// TIA Portal V16 export
// export: Created 2022-07-21T09:35:15.7704888Z, ExportSetting WithDefaults, DisplayName Totally Integrated Automation Portal, DisplayVersion V16 Update 4, DisplayName TIA Portal Version Control Interface, DisplayVersion V16 Update 2, DisplayName TIA Portal Openness, DisplayVersion V16 Update 4, DisplayName SINAMICS Startdrive Advanced, DisplayVersion V16 Update 5, DisplayName SINAMICS Startdrive G130, G150, S120, S150, SINAMICS MV, S210, DisplayVersion V16 Update 5, DisplayName SINAMICS Startdrive G110M, G120, G120C, G120D, G120P, G115D, DisplayVersion V16 Update 5, DisplayName STEP 7 Professional, DisplayVersion V16 Update 4, DisplayName STEP 7 Safety, DisplayVersion V16, DisplayName WinCC Advanced, DisplayVersion V16 Update 4
DATA_BLOCK "LAxisBasics_InterfaceHMI_3"   // DB843
{ S7_Optimized_Access := 'TRUE' }
AUTHOR : ArSc
FAMILY : LAxisBasics
VERSION : 1.1
// stored: AutoNumber false, DBAccessibleFromOPCUA true, InstanceOfName LAxisBasics_typeInterfaceHMI, InstanceOfType UDT, IsOnlyStoredInLoadMemory false, IsWriteProtectedInAS false
"LAxisBasics_typeInterfaceHMI"
   // VAR RETAIN
   //    axisDataToHMI { S7_SetPoint := 'True'} : "LAxisBasics_typeAxisDataToHMI";   // Panel 3
   // END_VAR
BEGIN
END_DATA_BLOCK
